{attribute 'GeneratedUsingTerminal: EL6201-0000-0017'}
{attribute addProperty BoxType "EL6201-0000-0017"}
{attribute addProperty Id "Slave_17A_DO0BOOL1Slave_17A_DO1BOOL1Slave_17A_DO2BOOL1Slave_17A_DO3BOOL1Slave_17B_DO0BOOL1Slave_17B_DO1BOOL1Slave_17B_DO2BOOL1Slave_17B_DO3BOOL1"}
{attribute addProperty CRC "1016142130"}
{attribute addProperty Size "8"}
TYPE Slave_17_Outputs_3C911932 :
STRUCT
	{attribute addProperty Name "Slave_17A_DO0"}
	Slave_17A_DO0 : BOOL;
	{attribute addProperty Name "Slave_17A_DO1"}
	Slave_17A_DO1 : BOOL;
	{attribute addProperty Name "Slave_17A_DO2"}
	Slave_17A_DO2 : BOOL;
	{attribute addProperty Name "Slave_17A_DO3"}
	Slave_17A_DO3 : BOOL;
	{attribute addProperty Name "Slave_17B_DO0"}
	Slave_17B_DO0 : BOOL;
	{attribute addProperty Name "Slave_17B_DO1"}
	Slave_17B_DO1 : BOOL;
	{attribute addProperty Name "Slave_17B_DO2"}
	Slave_17B_DO2 : BOOL;
	{attribute addProperty Name "Slave_17B_DO3"}
	Slave_17B_DO3 : BOOL;
END_STRUCT
END_TYPE

(* stored: Version 1.2.0.0, ProductVersion 3.1.4024.9
   DUT Slave_17_Outputs_3C911932: Id {566e33cf-1f5d-44e6-b23b-334635bfc9e1} *)
